FUNCTION_BLOCK CL_GreenhouseSystem extends CL_MasterRootClass
VAR_INPUT
END_VAR
VAR_OUTPUT
END_VAR
VAR
  nLastStateMachine         : E_StateMachine;
  nHistoStateMachine_AR     : ARRAY[0..100]OF E_StateMachine;
  //z                         : UINT;
  
  //INTERNAL VAR
  _nRequestModeMachine      : E_ModeMachine := E_ModeMachine.Automatic;
  _nModeMachine             : E_ModeMachine := E_ModeMachine.Automatic;
  _nStateMachine            : E_StateMachine := E_StateMachine.cIdle;
END_VAR

//State machine histroy
IF nLastStateMachine <> nStateMachine THEN
  nLastStateMachine := nStateMachine;  
  Case01Hysto(nStateMachine);
END_IF

//Manage Mode machine
IF _nRequestModeMachine <> nModeMachine AND _nStateMachine = E_StateMachine.cStopped THEN
	_nModeMachine := _nRequestModeMachine;
END_IF

PROPERTY nModeMachine : E_ModeMachine
GET
nModeMachine := _nModeMachine;
END_GET
SET
_nModeMachine := nModeMachine;
END_SET
END_PROPERTY

PROPERTY nStateMachine : E_StateMachine
GET
nStateMachine := _nStateMachine;
END_GET
SET
_nStateMachine := nStateMachine;
END_SET
END_PROPERTY

METHOD ReqModeMachine : BOOL
VAR_INPUT
  nModeMachine   :E_ModeMachine;
END_VAR
_nRequestModeMachine := nModeMachine;
END_METHOD

END_FUNCTION_BLOCK

(* stored: Version 1.1.0.1, ProductVersion 3.1.4024.12
   POU CL_GreenhouseSystem: Id {649a3c98-cef9-49ef-abcc-66e50a4447d0}, SpecialFunc None
   Property nModeMachine: Id {6ccbbe11-206f-4ece-886c-b3c198b618bd}
   Get Get: Id {e5d8187a-c430-43e9-aea1-e8db6ec3bf3e}
   Set Set: Id {274c2497-a6f8-4743-82d8-aaeef5ae1292}
   Property nStateMachine: Id {b22ca0d4-44a4-40c1-a42d-9361fd4d5108}
   Get Get: Id {5ff9b98b-39b3-4b78-a3b5-7b9e8ea604ac}
   Set Set: Id {a4bd60e8-afdc-4af0-a573-39811e224709}
   Method ReqModeMachine: Id {a96c1e55-f3b4-4370-a009-07d0ab47c4fc} *)
